// TIA Portal V21 export
VAR_GLOBAL   // PLC tag table "K_VistaManuale"
END_VAR
VAR_GLOBAL CONSTANT   // user constants
   K_VistaManuale_NessunaVista : Int := 0;
   K_VistaManuale_AltezzaStampo : Int := 1;
   K_VistaManuale_LameTaglioAltezza : Int := 2;
   K_VistaManuale_CaricoStecchi : Int := 3;
   K_VistaManuale_PreforaturaAghi : Int := 4;
   K_VistaManuale_RotazioneStampo : Int := 5;
   K_VistaManuale_SpintoreStecchi : Int := 6;
   "K_VistaManuale_CicloTaglio+Inserimento" : Int := 7;
END_VAR
